PROGRAM op_btn_ladder
VAR
END_VAR

// NETWORK 1

END_PROGRAM

(* stored: Version 1.1.0.1, ProductVersion 3.1.4024.12
   POU op_btn_ladder: Id {d85dcc85-c81f-4e0e-85e1-a80403bc43dc}, SpecialFunc None *)
